# EPICS substitutions: hyrel3dApp/Db/hyrel3d.substitutions
file hyrel3d.template
{ pattern { Sys		    , Dev,		    Yoke , Head  , PORT     , A		}
	  { "XF:11ID-M3" 	, "{Hyrel:1}",	1    , 2	 , "HYREL"  , 0	    }
}
